// SIMATIC STEP 7 (V5.x) project PLCSIM
// CPU: CPU 315-2 DP
// CPU: CPU 313
// CPU: CPU 412-1
// station: P_ADR_BUS
// station: Hardware
// station: SIMATIC 300(1)
// station: P_ADR_BUS
// station: Hardware
// station: SIMATIC 300(2)
// station: Hardware
// station: SIMATIC 400(1)
// station: P_ADR_BUS
// program: S7 Program(4)
// program: S7 Program(2)
// program: S7 Program(3)

SYMBOL_TABLE
"CYCL_EXC"	OB 1	OB 1	// Cycle Execution
"HW_INT0"	OB 40	OB 40	// Hardware Interrupt 0
"CYCL_FLT"	OB 80	OB 80	// Cycle Time Fault
"VAT_1"	VAT 1	
END_SYMBOL_TABLE

FUNCTION_BLOCK FB 1
VERSION : 0.1
VAR_INPUT
  pol1 : INT ;
  pol2 : INT ;
END_VAR
VAR_OUTPUT
  kv1 : BOOL ;
  kn1 : BOOL ;
  kv2 : BOOL ;
  kn2 : BOOL ;
END_VAR
BEGIN
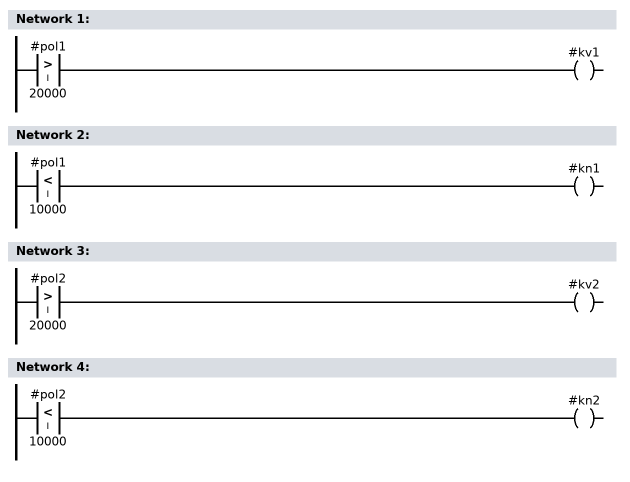
NETWORK
TITLE =
      L     #pol1;
      L     20000;
      >I;
      =     #kv1;
NETWORK
TITLE =
      L     #pol1;
      L     10000;
      <I;
      =     #kn1;
NETWORK
TITLE =
      L     #pol2;
      L     20000;
      >I;
      =     #kv2;
NETWORK
TITLE =
      L     #pol2;
      L     10000;
      <I;
      =     #kn2;
END_FUNCTION_BLOCK

FUNCTION FC 1 : VOID
VERSION : 0.1
VAR_INPUT
  in1 : INT ;
  in2 : INT ;
END_VAR
VAR_OUTPUT
  out1 : INT ;
  out2 : INT ;
END_VAR
BEGIN
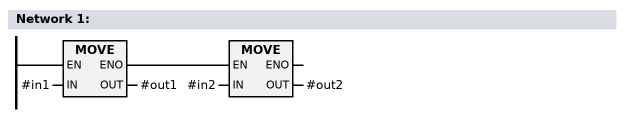
NETWORK
TITLE =
      A(;
      L     #in1;
      T     #out1;
      SET;
      SAVE;
      CLR;
      A     BR;
      );
      JNB   _001;
      L     #in2;
      T     #out2;
_001: NOP   0;
END_FUNCTION

DATA_BLOCK DB 1
VERSION : 0.1
  STRUCT
   pol1 : INT ;	//Temporary placeholder variable
   pol2 : INT ;
  END_STRUCT ;	
BEGIN
END_DATA_BLOCK

DATA_BLOCK DB 2
VERSION : 0.0
FB 1
BEGIN
END_DATA_BLOCK

ORGANIZATION_BLOCK "CYCL_EXC"	// OB 1
TITLE = "Main Program Sweep (Cycle)"
VERSION : 0.1
VAR_TEMP
  OB1_EV_CLASS : BYTE ;	//Bits 0-3 = 1 (Coming event), Bits 4-7 = 1 (Event class 1)
  OB1_SCAN_1 : BYTE ;	//1 (Cold restart scan 1 of OB 1), 3 (Scan 2-n of OB 1)
  OB1_PRIORITY : BYTE ;	//Priority of OB Execution
  OB1_OB_NUMBR : BYTE ;	//1 (Organization block 1, OB1)
  OB1_RESERVED_1 : BYTE ;	//Reserved for system
  OB1_RESERVED_2 : BYTE ;	//Reserved for system
  OB1_PREV_CYCLE : INT ;	//Cycle time of previous OB1 scan (milliseconds)
  OB1_MIN_CYCLE : INT ;	//Minimum cycle time of OB1 (milliseconds)
  OB1_MAX_CYCLE : INT ;	//Maximum cycle time of OB1 (milliseconds)
  OB1_DATE_TIME : DATE_AND_TIME ;	//Date and time OB1 started
END_VAR
BEGIN
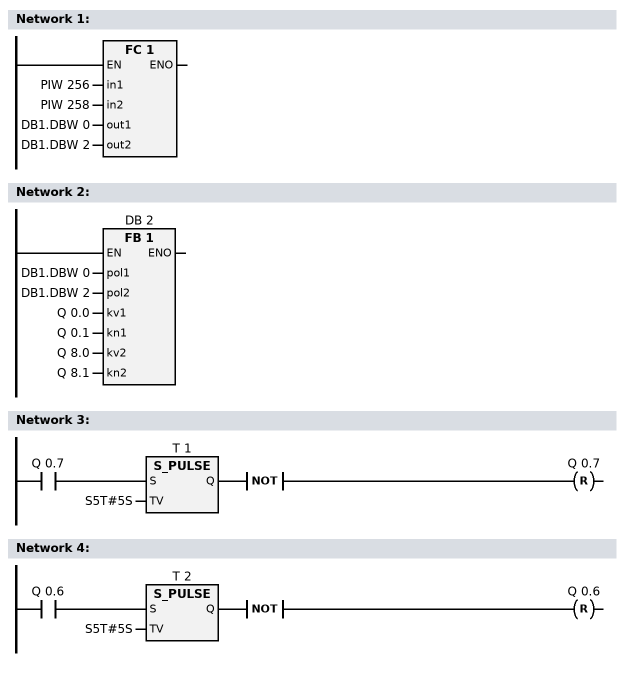
NETWORK
TITLE =
      CALL  FC 1 (
           in1                      := PIW 256,
           in2                      := PIW 258,
           out1                     := DB1.DBW 0,
           out2                     := DB1.DBW 2);
      NOP   0;
NETWORK
TITLE =
      CALL  FB 1 , DB 2 (
           pol1                     := DB1.DBW 0,
           pol2                     := DB1.DBW 2,
           kv1                      := Q 0.0,
           kn1                      := Q 0.1,
           kv2                      := Q 8.0,
           kn2                      := Q 8.1);
      NOP   0;
NETWORK
TITLE =
      A(;
      A     Q 0.7;
      L     S5T#5S;
      SP    T 1;
      NOP   0;
      NOP   0;
      NOP   0;
      A     T 1;
      );
      NOT;
      R     Q 0.7;
NETWORK
TITLE =
      A(;
      A     Q 0.6;
      L     S5T#5S;
      SP    T 2;
      NOP   0;
      NOP   0;
      NOP   0;
      A     T 2;
      );
      NOT;
      R     Q 0.6;
END_ORGANIZATION_BLOCK

ORGANIZATION_BLOCK "HW_INT0"	// OB 40
TITLE = "Hardware Interrupt"
VERSION : 0.1
VAR_TEMP
  OB40_EV_CLASS : BYTE ;	//Bits 0-3 = 1 (Coming event), Bits 4-7 = 1 (Event class 1)
  OB40_STRT_INF : BYTE ;	//16#41 (OB 40 has started)
  OB40_PRIORITY : BYTE ;	//Priority of OB Execution
  OB40_OB_NUMBR : BYTE ;	//40 (Organization block 40, OB40)
  OB40_RESERVED_1 : BYTE ;	//Reserved for system
  OB40_IO_FLAG : BYTE ;	//16#54 (input module), 16#55 (output module)
  OB40_MDL_ADDR : WORD ;	//Base address of module initiating interrupt
  OB40_POINT_ADDR : DWORD ;	//Interrupt status of the module
  OB40_DATE_TIME : DATE_AND_TIME ;	//Date and time OB40 started
END_VAR
BEGIN
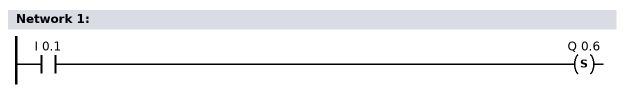
NETWORK
TITLE =
      A     I 0.1;
      S     Q 0.6;
END_ORGANIZATION_BLOCK

ORGANIZATION_BLOCK "CYCL_FLT"	// OB 80
TITLE = "Cycle Time Fault"
VERSION : 0.1
VAR_TEMP
  OB80_EV_CLASS : BYTE ;	//16#35, Event class 3, Entering event state, Internal fault event
  OB80_FLT_ID : BYTE ;	//16#XX, Fault identifcation code
  OB80_PRIORITY : BYTE ;	//Priority of OB Execution
  OB80_OB_NUMBR : BYTE ;	//80 (Organization block 80, OB80)
  OB80_RESERVED_1 : BYTE ;	//Reserved for system
  OB80_RESERVED_2 : BYTE ;	//Reserved for system
  OB80_ERROR_INFO : WORD ;	//Error information on event
  OB80_ERR_EV_CLASS : BYTE ;	//Class of event causing error
  OB80_ERR_EV_NUM : BYTE ;	//Number of event causing error
  OB80_OB_PRIORITY : BYTE ;	//Priority of OB causing error
  OB80_OB_NUM : BYTE ;	//Number of OB causing error
  OB80_DATE_TIME : DATE_AND_TIME ;	//Date and time OB80 started
END_VAR
BEGIN
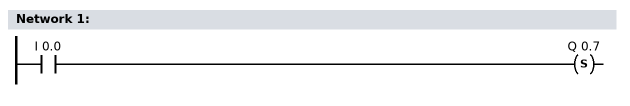
NETWORK
TITLE =
      A     I 0.0;
      S     Q 0.7;
END_ORGANIZATION_BLOCK

SYMBOL_TABLE
"M0.7"	M 0.7	BOOL
"VAT_"	VAT 1	
END_SYMBOL_TABLE

FUNCTION FC 1 : VOID
VERSION : 0.1
BEGIN
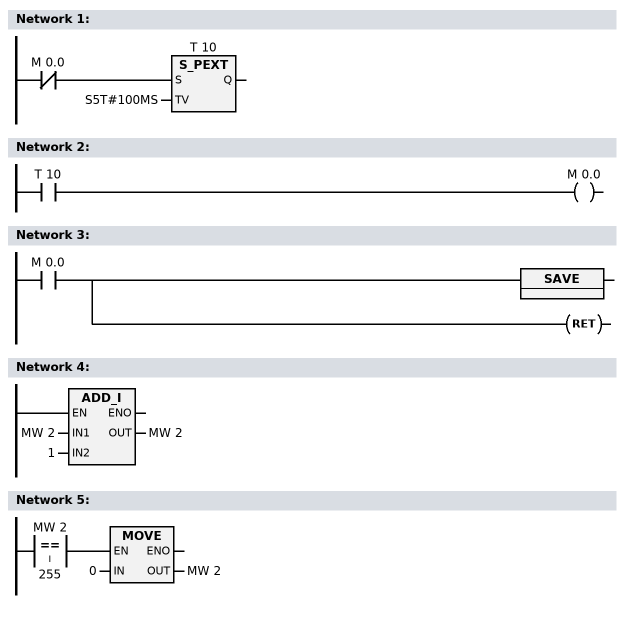
NETWORK
TITLE =
//далее идут фрагменты, реализующие тактовый байт 
      AN    M 0.0;
      L     S5T#100MS;
      SE    T 10;
      NOP   0;
      NOP   0;
      NOP   0;
      NOP   0;
NETWORK
TITLE =
      A     T 10;
      =     M 0.0;
NETWORK
TITLE =
      A     M 0.0;
      SAVE;
      BEC;
NETWORK
TITLE =
      L     MW 2;
      L     1;
      +I;
      T     MW 2;
      NOP   0;
NETWORK
TITLE =
      A(;
      L     MW 2;
      L     255;
      ==I;
      );
      JNB   _001;
      L     0;
      T     MW 2;
_001: NOP   0;
END_FUNCTION

ORGANIZATION_BLOCK OB 1
TITLE = "Main Program Sweep (Cycle)"
VERSION : 0.1
VAR_TEMP
  OB1_EV_CLASS : BYTE ;	//Bits 0-3 = 1 (Coming event), Bits 4-7 = 1 (Event class 1)
  OB1_SCAN_1 : BYTE ;	//1 (Cold restart scan 1 of OB 1), 3 (Scan 2-n of OB 1)
  OB1_PRIORITY : BYTE ;	//Priority of OB Execution
  OB1_OB_NUMBR : BYTE ;	//1 (Organization block 1, OB1)
  OB1_RESERVED_1 : BYTE ;	//Reserved for system
  OB1_RESERVED_2 : BYTE ;	//Reserved for system
  OB1_PREV_CYCLE : INT ;	//Cycle time of previous OB1 scan (milliseconds)
  OB1_MIN_CYCLE : INT ;	//Minimum cycle time of OB1 (milliseconds)
  OB1_MAX_CYCLE : INT ;	//Maximum cycle time of OB1 (milliseconds)
  OB1_DATE_TIME : DATE_AND_TIME ;	//Date and time OB1 started
END_VAR
BEGIN
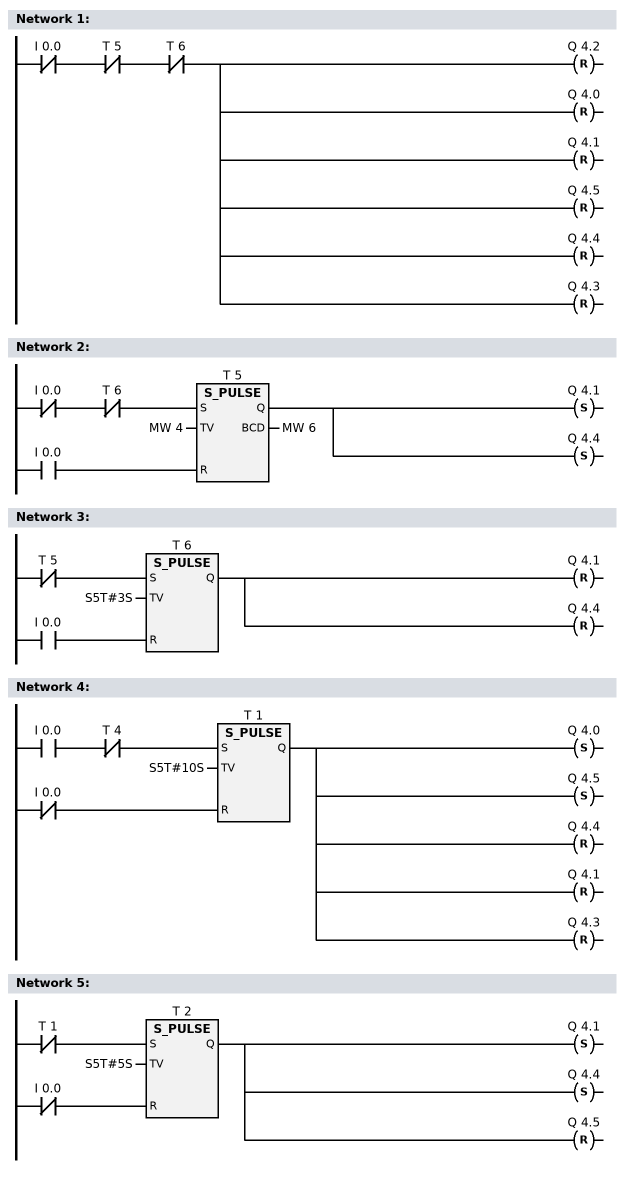
NETWORK
TITLE =
      AN    I 0.0;
      AN    T 5;
      AN    T 6;
      R     Q 4.2;
      R     Q 4.0;
      R     Q 4.1;
      R     Q 4.5;
      R     Q 4.4;
      R     Q 4.3;
NETWORK
TITLE =
      AN    I 0.0;
      AN    T 6;
      L     MW 4;
      SP    T 5;
      A     I 0.0;
      R     T 5;
      NOP   0;
      LC    T 5;
      T     MW 6;
      A     T 5;
      S     Q 4.1;
      S     Q 4.4;
NETWORK
TITLE =
      AN    T 5;
      L     S5T#3S;
      SP    T 6;
      A     I 0.0;
      R     T 6;
      NOP   0;
      NOP   0;
      A     T 6;
      R     Q 4.1;
      R     Q 4.4;
NETWORK
TITLE =
      A     I 0.0;
      AN    T 4;
      L     S5T#10S;
      SP    T 1;
      AN    I 0.0;
      R     T 1;
      NOP   0;
      NOP   0;
      A     T 1;
      S     Q 4.0;
      S     Q 4.5;
      R     Q 4.4;
      R     Q 4.1;
      R     Q 4.3;
NETWORK
TITLE =
      AN    T 1;
      L     S5T#5S;
      SP    T 2;
      AN    I 0.0;
      R     T 2;
      NOP   0;
      NOP   0;
      A     T 2;
      S     Q 4.1;
      S     Q 4.4;
      R     Q 4.5;
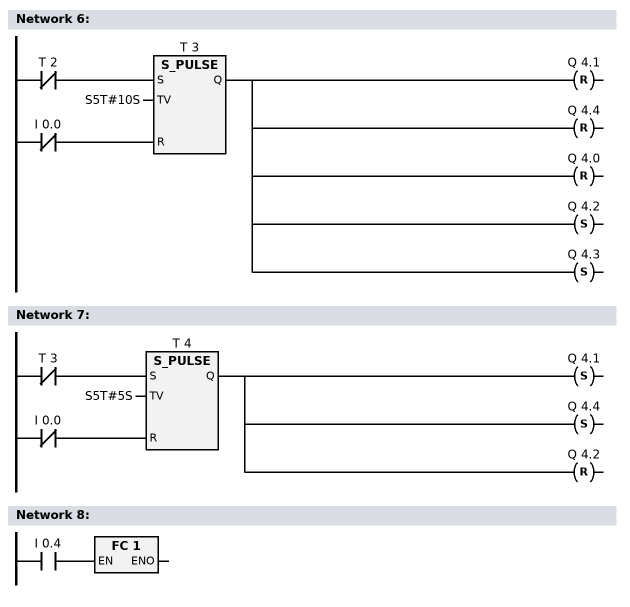
NETWORK
TITLE =
      AN    T 2;
      L     S5T#10S;
      SP    T 3;
      AN    I 0.0;
      R     T 3;
      NOP   0;
      NOP   0;
      A     T 3;
      R     Q 4.1;
      R     Q 4.4;
      R     Q 4.0;
      S     Q 4.2;
      S     Q 4.3;
NETWORK
TITLE =
      AN    T 3;
      L     S5T#5S;
      SP    T 4;
      AN    I 0.0;
      R     T 4;
      NOP   0;
      NOP   0;
      A     T 4;
      S     Q 4.1;
      S     Q 4.4;
      R     Q 4.2;
NETWORK
TITLE =
//Вызов функции, реализующей тактовый байт.
      A     I 0.4;
      JNB   _001;
      CALL  FC 1;
_001: NOP   0;
END_ORGANIZATION_BLOCK

SYMBOL_TABLE
"VAT_1"	VAT 1	
END_SYMBOL_TABLE

ORGANIZATION_BLOCK OB 1
TITLE = "Main Program Sweep (Cycle)"
VERSION : 0.1
VAR_TEMP
  OB1_EV_CLASS : BYTE ;	//Bits 0-3 = 1 (Coming event), Bits 4-7 = 1 (Event class 1)
  OB1_SCAN_1 : BYTE ;	//1 (Cold restart scan 1 of OB 1), 3 (Scan 2-n of OB 1)
  OB1_PRIORITY : BYTE ;	//Priority of OB Execution
  OB1_OB_NUMBR : BYTE ;	//1 (Organization block 1, OB1)
  OB1_RESERVED_1 : BYTE ;	//Reserved for system
  OB1_RESERVED_2 : BYTE ;	//Reserved for system
  OB1_PREV_CYCLE : INT ;	//Cycle time of previous OB1 scan (milliseconds)
  OB1_MIN_CYCLE : INT ;	//Minimum cycle time of OB1 (milliseconds)
  OB1_MAX_CYCLE : INT ;	//Maximum cycle time of OB1 (milliseconds)
  OB1_DATE_TIME : DATE_AND_TIME ;	//Date and time OB1 started
END_VAR
BEGIN
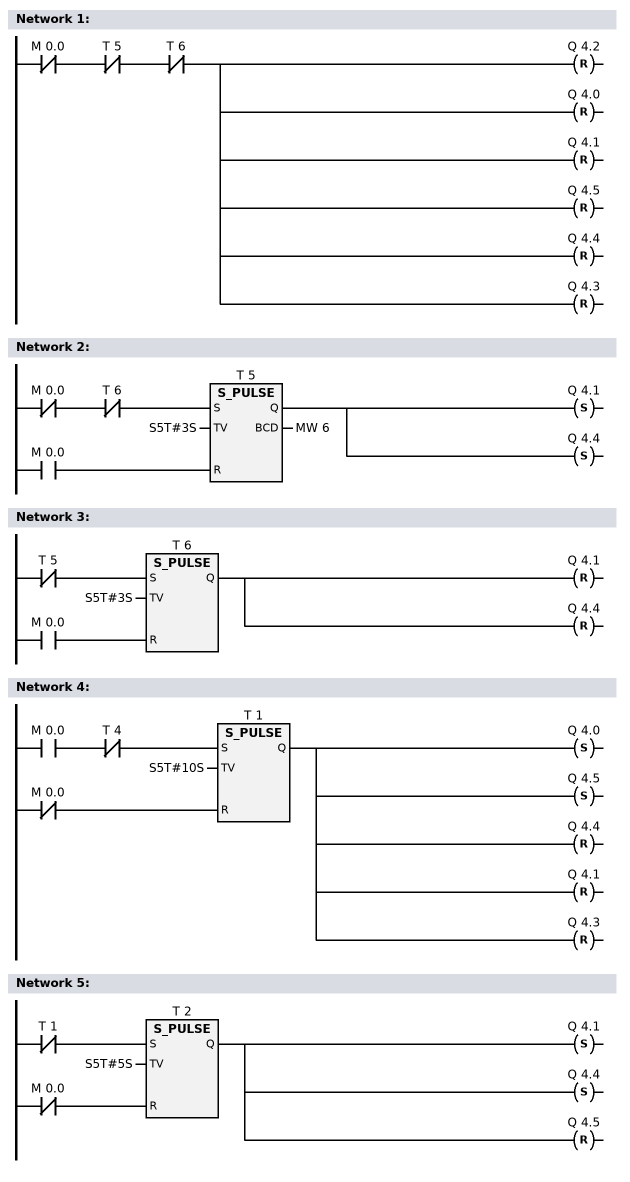
NETWORK
TITLE =
      AN    M 0.0;
      AN    T 5;
      AN    T 6;
      R     Q 4.2;
      R     Q 4.0;
      R     Q 4.1;
      R     Q 4.5;
      R     Q 4.4;
      R     Q 4.3;
NETWORK
TITLE =
      AN    M 0.0;
      AN    T 6;
      L     S5T#3S;
      SP    T 5;
      A     M 0.0;
      R     T 5;
      NOP   0;
      LC    T 5;
      T     MW 6;
      A     T 5;
      S     Q 4.1;
      S     Q 4.4;
NETWORK
TITLE =
      AN    T 5;
      L     S5T#3S;
      SP    T 6;
      A     M 0.0;
      R     T 6;
      NOP   0;
      NOP   0;
      A     T 6;
      R     Q 4.1;
      R     Q 4.4;
NETWORK
TITLE =
      A     M 0.0;
      AN    T 4;
      L     S5T#10S;
      SP    T 1;
      AN    M 0.0;
      R     T 1;
      NOP   0;
      NOP   0;
      A     T 1;
      S     Q 4.0;
      S     Q 4.5;
      R     Q 4.4;
      R     Q 4.1;
      R     Q 4.3;
NETWORK
TITLE =
      AN    T 1;
      L     S5T#5S;
      SP    T 2;
      AN    M 0.0;
      R     T 2;
      NOP   0;
      NOP   0;
      A     T 2;
      S     Q 4.1;
      S     Q 4.4;
      R     Q 4.5;
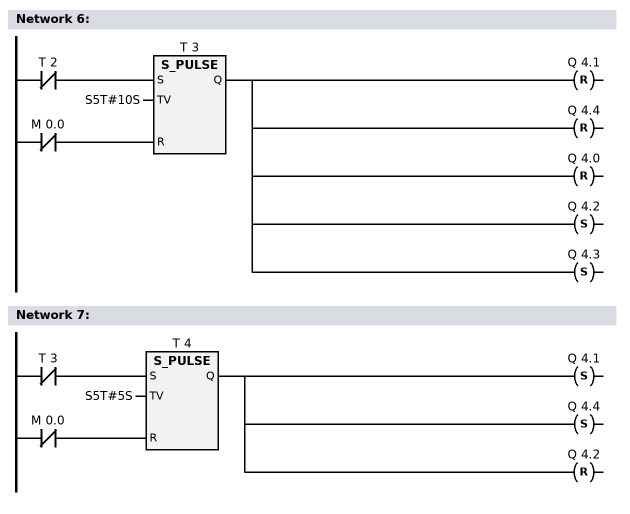
NETWORK
TITLE =
      AN    T 2;
      L     S5T#10S;
      SP    T 3;
      AN    M 0.0;
      R     T 3;
      NOP   0;
      NOP   0;
      A     T 3;
      R     Q 4.1;
      R     Q 4.4;
      R     Q 4.0;
      S     Q 4.2;
      S     Q 4.3;
NETWORK
TITLE =
      AN    T 3;
      L     S5T#5S;
      SP    T 4;
      AN    M 0.0;
      R     T 4;
      NOP   0;
      NOP   0;
      A     T 4;
      S     Q 4.1;
      S     Q 4.4;
      R     Q 4.2;
NETWORK
TITLE =
      A(;
      A     T 5;
      CU    C 1;
      BLD   101;
      NOP   0;
      NOP   0;
      A     M 0.0;
      R     C 1;
      L     C 1;
      T     MW 2;
      NOP   0;
      A     C 1;
      );
      A(;
      L     MW 2;
      L     5;
      >=I;
      );
      S     M 0.0;
NETWORK
TITLE =
      A(;
      A     T 1;
      CU    C 2;
      BLD   101;
      NOP   0;
      NOP   0;
      AN    M 0.0;
      R     C 2;
      L     C 2;
      T     MW 4;
      NOP   0;
      A     C 2;
      );
      A(;
      L     MW 4;
      L     5;
      >=I;
      );
      R     M 0.0;
END_ORGANIZATION_BLOCK
